Staubli VAL3: onF8Event.pgx

program onF8Event()
  local num x_nResult
begin
  // look if the bButton is enable
  if bButton[7]
    //
  endIf
end
